// TwinCAT 3 PLC project PLC01
// ProgramVersion: 3.1.4023.0
// libraries:
//   Tc2_ControllerToolbox, * (Beckhoff Automation GmbH)
//   Tc2_Standard, * (Beckhoff Automation GmbH)
//   Tc2_System, * (Beckhoff Automation GmbH)
//   Tc2_TempController, * (Beckhoff Automation GmbH)
//   Tc3_Module, * (Beckhoff Automation GmbH)
//   VisuDialogs, * (System)
// project tree:
//   DUTs/ stAutoTunningDef.TcDUT
//   / GlobalTextList.TcGTLO, PlcTask.TcTTO, Visualization Manager.TcVMO (not stored)
//   POUs/ FB_Blink.TcPOU, MAIN.TcPOU
//   VISUs/ ExtraParams.TcVIS, Footer.TcVIS, Visualization.TcVIS
// real-time tasks:
//   TASK PlcTask: cycle T#10ms, priority 20, ADS port 350
//   TASK PlcTask1: cycle T#10ms, priority 21, ADS port 351
// variable links:
//   PLC01 Instance <-> Simulation/Simulation Instance
//     PlcTask Inputs/MAIN.currTemp <-> PlcTask Outputs/MAIN.actualTemp
//     PlcTask Outputs/MAIN.fyAnalogOutput <-> PlcTask Inputs/MAIN.tempCmd

CONFIGURATION PLC01
    RESOURCE PLC ON TwinCAT3
        TASK PlcTask(INTERVAL := T#10ms, PRIORITY := 20);
        PROGRAM MAIN WITH PlcTask : MAIN;
    END_RESOURCE
END_CONFIGURATION

// ---- DUTs/stAutoTunningDef.TcDUT
TYPE stAutoTunningDef :
STRUCT
	fTuneKp:LREAL;
	fTuneTn:LREAL;
	fTuneTv:LREAL;
	fTuneTd:LREAL;
END_STRUCT
END_TYPE

// ---- POUs/MAIN.TcPOU
PROGRAM MAIN
VAR
	controller:FB_CTRL_TempController;
	tempSetpoint:ARRAY[1..2] OF LREAL:=[100,50];
	currTemp AT %I*:LREAL;
	fyAnalogOutput AT %Q*:LREAL;
	bSelSetpoint: BOOL;
	eCtrlMode: E_CTRL_MODE := E_CTRL_MODE.eCTRL_MODE_IDLE;
	eCtrlState: Tc2_TempController.E_CTRL_STATE;
	internalParams: Tc2_TempController.ST_CTRL_ParaController;
	startTunning: BOOL;

	activeSetpoint: LREAL;
	bCopyParams:BOOL;	//copy internal params into external params
	startAutoTunning: BOOL;
	bStartCtrlAfterTunning: BOOL;
	trigTunningFinished:R_TRIG;

	bErrorActive: BOOL;
	errId: Tc2_TempController.E_CTRL_ErrorCodes;
	bOutputHeat: BOOL;
	bOutputCool: BOOL;
	blink:FB_Blink;
	blinkLed: BOOL;
	bBlinkError: BOOL;
	iTunningType:INT;
	startController: BOOL;
	stopController: BOOL;
END_VAR
VAR PERSISTENT
	externalParams: ST_CTRL_ParaController;
	stControllerParameter	: ST_CTRL_TempCtrlParameter := (		
		
		(* general parameters 													 *)
		iMode					:= 1,											(* 1=heating, 2=cooling, 3=heating&cooling *)
		iReactionOnFailure		:= eCTRL_ReactionOnFailure_StopController,		(* 0=controller off, 1=manual op, 2=yMin, 3=yMax *)
	
		bSelCtrlParameterSet	:= FALSE,										(* FALSE = internal set, TRUE = external set *)
	
		dwAlarmSupp				:= 16#0000EFFF,									(* alarm suppression *)
		tCtrlCycleTime			:= T#500MS,										(* controller cycle time *)
		tTaskCycleTime			:= T#10MS,										(* plc task cycle time *)
		
		(* tuning parameters 													 *)
		iTuningMode				:= 1,											(* only heating, only cooling, first heating then cooling or vice versa *)
	
		tTuneStabilisation		:= T#20S,										(* wait for a stable system *)
	
		fEndTunePercentHeating	:= 80.0,										(* switch to closed loop control when X > 0.8*W *)
		fYTuneHeating			:= 100.0,										(* step change while tuning operation *)
		fYStableHeating			:= 0.0,											(* tuning operation *)
	
		fEndTunePercentCooling	:= 20.0,										(* switch to closed loop control when X < 0.2*W *)
		fYTuneCooling			:= 0.0,											(* step change while tuning operation *)
		fYStableCooling			:= 0.0,											(* tuning operation *)
		fScalingFactor			:= 1.0,											(* Scaling factor for KP heating/cooling *)
		
		(* setpoint parameters 													 *)
		fWMin					:= 0.0,											(* lower limit *)
		fWMax					:= 300.0,										(* upper limit *)
	
		(* start up *)
		bEnableSoftStart		:= FALSE,										(* FALSE = no soft start, TRUE = soft start *)
		bEnableRamping			:= FALSE,										(* FALSE = no ramping, TRUE = ramping *)
	
		fWStartUp				:= 0.0,											(* soft start plateau setpoint *)
		tStartUp				:= T#0MS,										(* soft start waiting time*)
		bStartUpRamping			:= FALSE,										(* enable ramping while start up phase *)
		fWStartUpVeloPos		:= 1.0,											(* max gradient for increasing setpoint in start up phase*)
		fWStartUpVeloNeg		:= 1.0,											(* max gradient for decreasing setpoint in start up phase *)
	
		fWVeloPos				:= 1.0,											(* max gradient for increasing setpoint *)
		fWVeloNeg				:= 1.0,											(* max gradient for decreasing setpoint *)	
	
		(* actual value parameters     											 *)
		bFilter 				:= FALSE,
		tFilter					:= T#0S,
		
		(* deadband parameters     												 *)
		bDeadband				:= FALSE,
		fEDeadband				:= 0.0,											(* deadband *)
		
		(* control value parameters     										 *)
		fYMin					:= 0.0,											(* lower limit *)
		fYMax					:= 100.0,										(* upper limit *)
		fYManual				:= 0.0,									 		(* manual operation*)
		fYOnFailure				:= 0.0,											(* control value on failure *)
	
		tPWMCycleTime			:= t#1s,										(* PWM: period *)
		tPWMMinOffTime			:= t#0s,										(* PWM: min off time *)
		tPWMMinOnTime			:= t#0s,										(* PWM: min on time *)
		tPWMWaitingTime			:= t#0s,										(* PWM: min waiting time *) (* not yet implemented !!!!*)
	
		fYThresholdOff			:= 0.0,											(* 3-Point: Off threshold *)
		fYThresholdOn			:= 0.0,											(* 3-Point: On threshold *)
	
		nCyclesForSwitchOver	:= 100,
	
		(* controller settings			     									 *)
		bEnablePreController 	:= FALSE,										(* enable precontroller *)
		bEnableZones 			:= FALSE,										(* enable zone around setpoint with open loop control *)
		bEnableCVFilter 		:= FALSE,										(* enable filter for CV (type see iFilterType) *)
		iFilterType 			:= E_FilterType_FIRSTORDER,			 			(* filtertype of CV filter *)
		iControllerType 		:= eCTRL_ControllerType_PID,					(* used controller normally PID *)
		
		
		(* min max temperatures	     											 *)
		TempLow					:= -5.0,
		TempLowLow				:= -10.0,
		TempHigh				:= 5.0,
		TempHighHigh			:= 10.0,
		TempAbsoluteHigh		:= 300.0,
		TempAbsoluteLow			:= 0.0,	
		
		(* internal tuning parameters *)
		fTuneKp					:= 1.2,
		fTuneTn					:= 2.0,
		fTuneTv					:= 0.42,
		fTuneTd					:= 0.25
		);
		softStartWaitTime:LREAL;
END_VAR
VAR CONSTANT
	aTuneDefParams: ARRAY [0..2] OF stAutoTunningDef := [(fTuneKp := 1.2, fTuneTn := 2.0, fTuneTv := 0.42, fTuneTd := 0.25), (fTuneKp := 1.0, fTuneTn := 2.5, fTuneTv := 0.42, fTuneTd := 0.25), (fTuneKp := 0.5, fTuneTn := 3.0, fTuneTv := 1.0, fTuneTd := 0.25)];
END_VAR

actModeMgmt();

trigTunningFinished(CLK:= eCtrlState = E_CTRL_STATE.eCTRL_STATE_TUNED);
IF trigTunningFinished.Q AND bStartCtrlAfterTunning THEN
	eCtrlMode:= E_CTRL_MODE.eCTRL_MODE_ACTIVE;
END_IF

controller(
	eCtrlMode:=eCtrlMode , 
	bSelSetpoint:= bSelSetpoint, 
	fW1:=tempSetpoint[1] , 
	fW2:= tempSetpoint[2], 
	fX:= currTemp, 
	fYManual:= , 
	sParaControllerExternal:= externalParams, 
	sControllerParameter:=stControllerParameter, 
	fYAnalog=> fyAnalogOutput, 
	eCtrlState=> eCtrlState, 
	sParaControllerInternal=> internalParams, 
	bError=>bErrorActive , 
	eErrorId=> errId);
	
actValueCopy();

bBlinkError:= bErrorActive AND blinkLed;

blink(timeOn:= T#500MS, timeOff:= T#700MS, bOutput=>blinkLed );

ACTION actModeMgmt:
IF startAutoTunning AND eCtrlState <> E_CTRL_STATE.eCTRL_STATE_TUNING AND eCtrlState <> E_CTRL_STATE.eCTRL_STATE_TUNED AND 
	eCtrlState <> E_CTRL_STATE.eCTRL_STATE_ERROR AND eCtrlState <> E_CTRL_STATE.eCTRL_STATE_RESET THEN
	eCtrlMode:= E_CTRL_MODE.eCTRL_MODE_TUNE;
END_IF


IF startController AND eCtrlState <> E_CTRL_STATE.eCTRL_STATE_TUNING AND eCtrlState <> E_CTRL_STATE.eCTRL_STATE_ERROR THEN
	eCtrlMode:= E_CTRL_MODE.eCTRL_MODE_ACTIVE;
END_IF

IF stopController THEN
	eCtrlMode:= E_CTRL_MODE.eCTRL_MODE_IDLE;
END_IF
END_ACTION

ACTION actValueCopy:
IF bCopyParams THEN
	externalParams:=internalParams;
END_IF

bOutputHeat:=controller.bYPWMPos;
bOutputCool:=controller.bYPWMNeg;

IF iTunningType >=0 AND iTunningType<=2 THEN
	stControllerParameter.fTuneKp:=aTuneDefParams[iTunningType].fTuneKp;
	stControllerParameter.fTuneTn:=aTuneDefParams[iTunningType].fTuneTn;
	stControllerParameter.fTuneTv:=aTuneDefParams[iTunningType].fTuneTv;
	stControllerParameter.fTuneTd:=aTuneDefParams[iTunningType].fTuneTd;
END_IF

activeSetpoint:=SEL(bSelSetpoint, tempSetpoint[1],tempSetpoint[2]);
stControllerParameter.tStartUp:= LREAL_TO_TIME(softStartWaitTime*1000);
END_ACTION

END_PROGRAM

// ---- POUs/FB_Blink.TcPOU
FUNCTION_BLOCK FB_Blink
VAR_INPUT
	timeOn:TIME:=T#300MS;
	timeOff:TIME:=T#500MS;
END_VAR
VAR_OUTPUT
	bOutput: BOOL;
END_VAR
VAR
	timer:TON;
END_VAR

timer(IN:= NOT timer.Q);
IF timer.Q THEN
	IF bOutput THEN
		timer.PT:=timeOff;
	ELSE
		timer.PT:=timeOn;	
	END_IF
	bOutput:= NOT bOutput;
END_IF

END_FUNCTION_BLOCK

// ---- GlobalTextList.TcGTLO
TEXTLIST GlobalTextList
  565 = '% Finish tunning'
  80 = '% Finish tunning cool'
  444 = '% Finish tunning heat'
  480 = '%.1'
  83 = '%.1F'
  366 = '%.1f'
  190 = '%d'
  695 = '%Finish tunning'
  830 = '%s'
  913 = '%t'
  75 = 'Auto-Tunning'
  891 = 'Checkbox'
  555 = 'Controller Off'
  135 = 'Controller On'
  87 = 'Controller output'
  289 = 'Controller state'
  675 = 'Copy intenal >> external'
  926 = 'Curr Temp.'
  79 = 'Curr. setpoint'
  818 = 'Error'
  972 = 'Error code'
  647 = 'External'
  890 = 'GroupBox'
  698 = 'Iniciar'
  977 = 'Internal'
  559 = 'Kp Cool'
  286 = 'Kp Heat'
  892 = 'Label'
  667 = 'MAIN'
  401 = 'Monitoring'
  672 = 'Output cool'
  1 = 'Output heat'
  511 = 'Param to use'
  465 = 'Parameters'
  942 = 'Parâmetros'
  88 = 'Principal'
  184 = 'Setpoint'
  392 = 'Setpoint 1'
  516 = 'Setpoint 2'
  900 = 'Setponit'
  865 = 'Soft Start'
  893 = 'Soft start temp'
  151 = 'Start'
  606 = 'Start control'
  634 = 'Start Ctrl after tunning'
  541 = 'Stop Control'
  922 = 'Td Cool'
  934 = 'Td Heat'
  938 = 'Tempo'
  222 = 'Tn Cool'
  681 = 'Tn Heat'
  273 = 'Tunning agressive'
  882 = 'Tunning fast'
  73 = 'Tunning medium'
  534 = 'Tunning no overshoot'
  485 = 'TV Cool'
  147 = 'Tv Cool'
  539 = 'TV Heat'
  113 = 'Tv Heat'
  367 = 'Use 2 setpoint'
  14 = 'Use External param set'
  347 = 'Use softstart'
  594 = 'When activated select the external params'
END_TEXTLIST

// ---- VISUs/ExtraParams.TcVIS
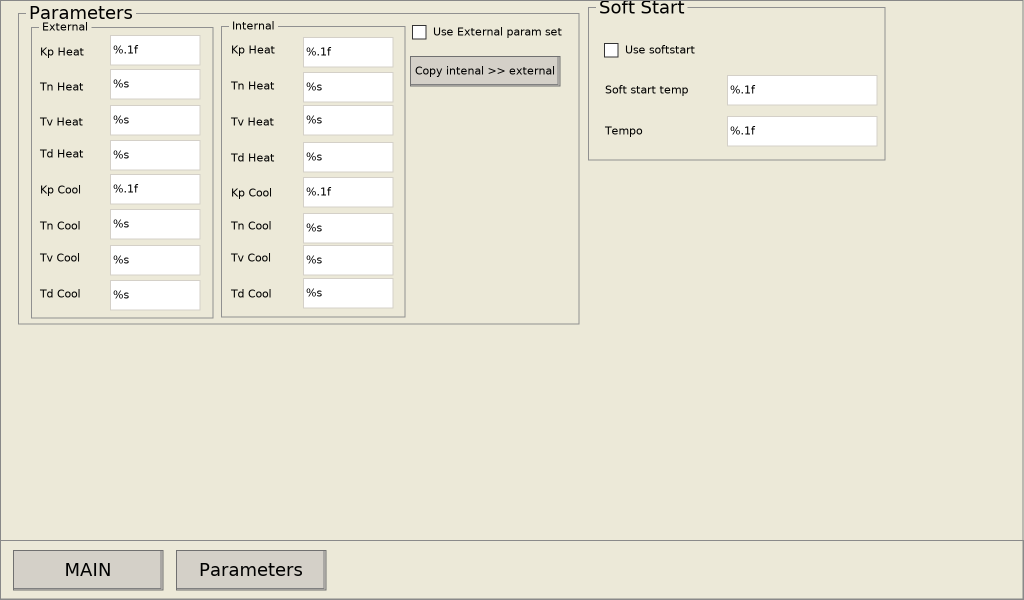
VISUALIZATION ExtraParams  // 1024x600
    GroupBox (18,5 561x319), "Parameters"
        GroupBox (13,14 182x299), "External"
            Label (6,18 70x30), "Kp Heat"
            Label (6,53 70x30), "Tn Heat"
            Label (6,88 70x30), "Tv Heat"
            Label (6,120 70x30), "Td Heat"
            Label (6,156 70x30), "Kp Cool"
            Label (6,192 70x30), "Tn Cool"
            Label (6,224 70x30), "Tv Cool"
            Label (6,260 70x30), "Td Cool"
            Textfield (79,16 90x30), "%.1f", text variable: MAIN.externalParams.KpHeat
            Textfield (79,50 90x30), "%s", text variable: MAIN.externalParams.TnHeat
            Textfield (79,86 90x30), "%s", text variable: MAIN.externalParams.TvHeat
            Textfield (79,121 90x30), "%s", text variable: MAIN.externalParams.TdHeat
            Textfield (79,155 90x30), "%.1f", text variable: MAIN.externalParams.KpCool
            Textfield (79,190 90x30), "%s", text variable: MAIN.externalParams.TnCool
            Textfield (79,226 90x30), "%s", text variable: MAIN.externalParams.TvCool
            Textfield (79,261 90x30), "%s", text variable: MAIN.externalParams.TdCool
        GroupBox (203,13 184x299), "Internal"
            Label (7,17 70x30), "Kp Heat"
            Label (7,53 70x30), "Tn Heat"
            Label (7,89 70x30), "Tv Heat"
            Label (7,125 70x30), "Td Heat"
            Label (7,160 70x30), "Kp Cool"
            Label (7,193 70x30), "Tn Cool"
            Label (7,225 70x30), "Tv Cool"
            Label (7,261 70x30), "Td Cool"
            Textfield (82,19 90x30), "%.1f", text variable: MAIN.internalParams.KpHeat
            Textfield (82,54 90x30), "%s", text variable: MAIN.internalParams.TnHeat
            Textfield (82,87 90x30), "%s", text variable: MAIN.internalParams.TvHeat
            Textfield (82,124 90x30), "%s", text variable: MAIN.internalParams.TdHeat
            Textfield (82,159 90x30), "%.1f", text variable: MAIN.internalParams.KpCool
            Textfield (82,195 90x30), "%s", text variable: MAIN.internalParams.TnCool
            Textfield (82,227 90x30), "%s", text variable: MAIN.internalParams.TvCool
            Textfield (82,260 90x30), "%s", text variable: MAIN.internalParams.TdCool
        Checkbox (392,12 172x30), "Use External param set", tooltip "When activated select the external params", variable: MAIN.stControllerParameter.bSelCtrlParameterSet
        Button (392,51 150x30), "Copy intenal >> external"
            tap MAIN.bCopyParams
    Frame (0,540 1024x60)
        shows Footer()
    GroupBox (588,-1 297x161), "Soft Start"
        Checkbox (14,36 116x30), "Use softstart", variable: MAIN.stControllerParameter.bEnableSoftStart
        Label (14,76 116x30), "Soft start temp"
        Textfield (139,76 150x30), "%.1f", text variable: MAIN.stControllerParameter.fWStartUp
            OnMouseClick: write the text variable via Default
        Label (14,117 100x30), "Tempo"
        Textfield (139,117 150x30), "%.1f", text variable: MAIN.softStartWaitTime
            OnMouseClick: write the text variable via Default
END_VISUALIZATION

// ---- VISUs/Footer.TcVIS
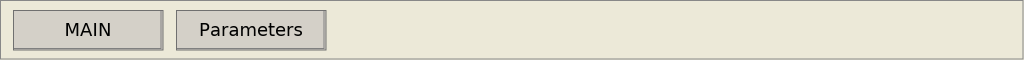
VISUALIZATION Footer  // 1024x60
    Button (13,10 150x40), "MAIN"
        OnMouseClick: change screen: Visualization
    Button (176,10 150x40), "Parameters"
        OnMouseClick: change screen: Footer
END_VISUALIZATION

// ---- VISUs/Visualization.TcVIS
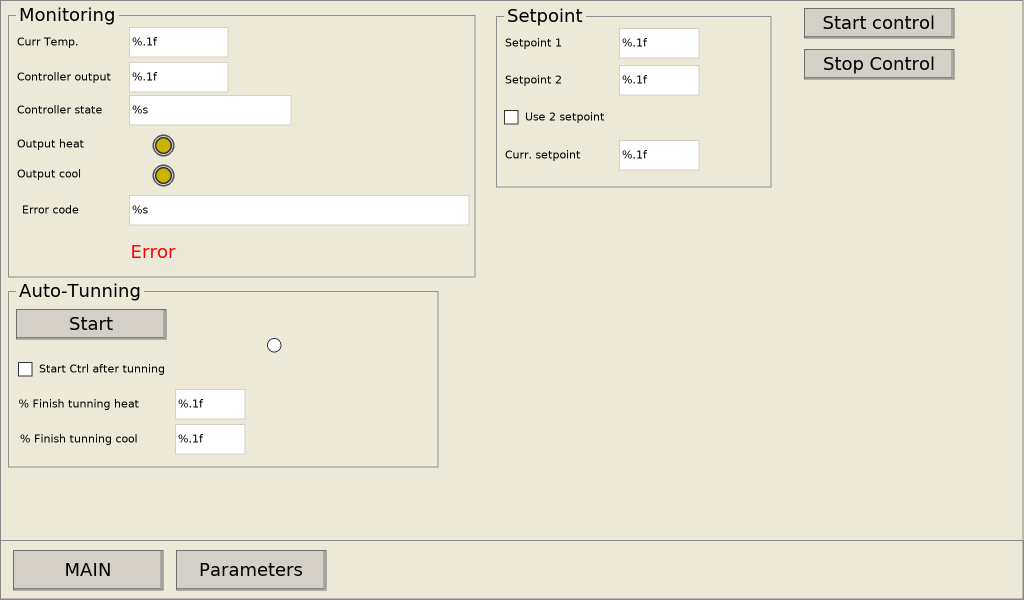
VISUALIZATION Visualization  // 1024x600
    GroupBox (496,8 275x179), "Setpoint"
        Checkbox (6,94 120x30), "Use 2 setpoint", variable: MAIN.bSelSetpoint
        Textfield (123,20 80x30), "%.1f", text variable: MAIN.tempSetpoint[1]
            OnMouseClick: write the text variable via Default
        Textfield (123,57 80x30), "%.1f", text variable: MAIN.tempSetpoint[2]
            OnMouseClick: write the text variable via Default
        Label (6,57 110x30), "Setpoint 2"
        Label (6,20 110x30), "Setpoint 1"
        Textfield (123,132 80x30), "%.1f", text variable: MAIN.activeSetpoint
        Label (6,132 110x30), "Curr. setpoint"
    GroupBox (8,7 467x270), "Monitoring"
        Textfield (121,20 99x30), "%.1f", text variable: MAIN.currTemp
        Textfield (121,88 162x30), "%s", text variable: MAIN.eCtrlState
        Label (6,88 110x30), "Controller state"
        Label (6,20 110x30), "Curr Temp."
        Textfield (121,55 99x30), "%.1f", text variable: MAIN.fyAnalogOutput
        Label (6,55 110x30), "Controller output"
        Label (6,122 160x30), "Output heat"
        Lamp1 (143,126 25x25), variable: MAIN.bOutputHeat, style: Lamp-Lamp1-Yellow
        Label (6,152 160x30), "Output cool"
        Textfield (121,188 340x30), "%s", text variable: MAIN.errId
        Label (93,230 104x30), "Error", invisible if: not MAIN.bBlinkError
    GroupBox (8,283 430x184), "Auto-Tunning"
        Button (8,26 150x30), "Start"
            tap MAIN.startAutoTunning
        Checkbox (8,71 163x30), "Start Ctrl after tunning", variable: MAIN.bStartCtrlAfterTunning
        Textfield (167,106 70x30), "%.1f", text variable: MAIN.stControllerParameter.fEndTunePercentHeating
            OnMouseClick: write the text variable via Default, min 10, max 90
        Label (6,106 130x30), "% Finish tunning heat"
        Textfield (167,141 70x30), "%.1f", text variable: MAIN.stControllerParameter.fEndTunePercentCooling
            OnMouseClick: write the text variable via Default, min 10, max 90
        RadioButton (257,15 169x94), variable: MAIN.iTunningType
            Areas[0]: Text=Tunning fast
            Areas[1]: Text=Tunning medium
            Areas[2]: Text=Tunning no overshoot
    Lamp1 (151,163 25x25), variable: MAIN.bOutputCool, style: Lamp-Lamp1-Yellow
    Label (19,195 104x30), "Error code"
    Label (14,424 130x30), "% Finish tunning cool"
    Button (804,8 150x30), "Start control"
        tap MAIN.startController
    Button (804,49 150x30), "Stop Control"
        tap MAIN.stopController
    Frame (0,540 1024x60)
        shows Footer()
END_VISUALIZATION
